(* PLC project Senza_nome, Sconosciuto Senza_nome 1 *)
(* stored: creationDateTime 2026-08-27T14:08:36, modificationDateTime 2026-08-27T14:18:28 *)

PROGRAM program0
  VAR
    bt1 : BOOL;
    reset : BOOL;
    OT_CV : INT;
    IN_PV : INT := 5;
    led : BOOL;
    CTU0 : CTU;
  END_VAR
  VAR  (* added by the conversion: wires and edge detectors of the diagram *)
    R_TRIG1 : R_TRIG;
  END_VAR

(* FBD diagram, written out as Structured Text *)
R_TRIG1(CLK := bt1);
CTU0(CU := R_TRIG1.Q, R := reset, PV := IN_PV);
led := CTU0.Q;
OT_CV := CTU0.CV;
END_PROGRAM

CONFIGURATION Config0
  RESOURCE Res0 ON PLC
    TASK task0(INTERVAL := T#20ms, PRIORITY := 0);
    PROGRAM instance0 WITH task0 : program0;
  END_RESOURCE
END_CONFIGURATION
